{attribute addProperty BoxType "AX8118-0100-0101-0101"}
{attribute addProperty Id "DeviceDevice_F82A60211620Device_SafetyDevice_Safety_AF71BE9D160200Ch_ACh_A_359CD49A176220WcStateAT %I*WcState_DC9C971540.50InfoDataAT %I*InfoData_F030DC9B200250"}
{attribute addProperty CRC "1051991048"}
{attribute addProperty SizeInBites "556"}
{attribute addProperty SizeInBytes "69.5"}
TYPE AX8118_E4DF8033 :
STRUCT
	{attribute addProperty Name "Device"}
	Device : Device_F82A6021;
	{attribute addProperty Name "Device_Safety"}
	Device_Safety : Device_Safety_AF71BE9D;
	{attribute addProperty Name "Ch_A"}
	Ch_A : Ch_A_359CD49A;
	{attribute addProperty Name "WcState"}
	WcState : WcState_DC9C9715;
	{attribute addProperty Name "InfoData"}
	InfoData : InfoData_F030DC9B;
END_STRUCT
END_TYPE

(* stored: Version 1.2.0.0, ProductVersion 3.1.4024.9
   DUT AX8118_E4DF8033: Id {f3010774-f261-4618-a3f7-133b0bde5783} *)
